TYPE ST_ComponentMyComponent_Status :
	STRUCT
		MyVarProperty1 : BOOL;
	END_STRUCT
END_TYPE

(* stored: Version 1.1.0.1, ProductVersion 3.1.4024.12
   DUT ST_ComponentMyComponent_Status: Id {4b8bc812-77af-4661-a312-32bb504738b3} *)
